INTERFACE I_CalibratableLinear EXTENDS I_Base

PROPERTY CalibrateLinear : I_CalibrateLinear
GET
END_GET
SET
END_SET
END_PROPERTY

END_INTERFACE

(* stored: Version 1.1.0.1, ProductVersion 3.1.4026.18
   Itf I_CalibratableLinear: Id {f8b48c81-d24c-4471-baf3-a0312f9c1f93}
   Property CalibrateLinear: Id {1132c595-aafb-477a-9959-f8a5a0ea0cf5}
   Get Get: Id {55d18c31-281d-4099-9a33-d60c826670f0}
   Set Set: Id {925796c2-b8a0-4f7e-b9eb-00d673331c40} *)
